// TIA Portal V20 export
DATA_BLOCK "LAF_InternalManual"   // DB43
VERSION : 19.0
// stored: MemoryReserve 100
   VAR
      hmi : Array[1..1] of "LAF_typeManHmiDisp";   // number of HMIs - modify the array size based on the required HMIs
      manualOperationEnabled : Bool;   // feedback whether the manual operation lines are selected
      emsWithManualOpConfigured { ExternalWritable := 'False'} : "LGM_emsWithManualOpConfigured";   // List of EMs with manual operation configured, for HMI button visibility
      disableUnit1 { S7_SetPoint := 'True'} : Bool;
      RisingEdge : Bool;
   END_VAR
BEGIN
END_DATA_BLOCK
